TYPE DUT_STRUCT_C000007_DEV :
STRUCT
	sCellName			:STRING := 'C0000007';
	sIpAddress			:STRING := '';
	sAmsNetId			:STRING := '';
	sOpcUaURL			:STRING := 'opc.tcp://:4840';
	sStation1			:STRING := 'S00000B';
END_STRUCT
END_TYPE

(* stored: Version 1.1.0.1, ProductVersion 3.1.4024.5
   DUT DUT_STRUCT_C000007_DEV: Id {eb6bd290-025d-41d1-8a0d-3e955aa12bde} *)
